PROGRAM Log_Diverts_P2150
VAR
	r_DivertExtend			: ARRAY [1..16] OF R_TRIG;
	f_DivertExtend			: ARRAY [1..16] OF F_TRIG;
	r_ConfirmPE				: ARRAY [1..16] OF R_TRIG;
	f_ConfirmPE				: ARRAY [1..16] OF F_TRIG;
	sMessage				: STRING;
END_VAR

// Divert 1
r_DivertExtend[1](CLK := Sorter.aSorterDiverts_P2150[1].Output1);
f_DivertExtend[1](CLK := Sorter.aSorterDiverts_P2150[1].Output1);

IF r_DivertExtend[1].Q THEN
	IF .nDivertLogEnable.DIVERT1 THEN
		ADSLOGSTR( msgCtrlMask := ADSLOG_MSGTYPE_HINT OR ADSLOG_MSGTYPE_LOG
			, msgFmtStr := 'Extend Divert 1 : %s'
			, strArg := UDINT_TO_STRING(Sorter.st_SorterEncoder_P2150.CurrentCount)); 
	END_IF;
END_IF
IF f_DivertExtend[1].Q THEN
	IF .nDivertLogEnable.DIVERT1 THEN
		ADSLOGSTR( msgCtrlMask := ADSLOG_MSGTYPE_HINT OR ADSLOG_MSGTYPE_LOG
			, msgFmtStr := 'Retract Divert 1 : %s'
			, strArg := UDINT_TO_STRING(Sorter.st_SorterEncoder_P2150.CurrentCount)); 
	END_IF;
END_IF

// Confirm 1
r_ConfirmPE[1](CLK := Sorter.aSorterDiverts_P2150[1].ConfirmPE);
f_ConfirmPE[1](CLK := Sorter.aSorterDiverts_P2150[1].ConfirmPE);

IF r_ConfirmPE[1].Q THEN
	IF .nDivertLogEnable.CONFIRM1 THEN
		ADSLOGSTR( msgCtrlMask := ADSLOG_MSGTYPE_HINT OR ADSLOG_MSGTYPE_LOG
			, msgFmtStr := 'Confirm PE 1 Blocked: %s'
			, strArg := UDINT_TO_STRING(Sorter.st_SorterEncoder_P2150.CurrentCount)); 
	END_IF;
END_IF
IF f_ConfirmPE[1].Q THEN
	IF .nDivertLogEnable.CONFIRM1 THEN
		ADSLOGSTR( msgCtrlMask := ADSLOG_MSGTYPE_HINT OR ADSLOG_MSGTYPE_LOG
			, msgFmtStr := 'Confirm PE 1 Clear: %s'
			, strArg := UDINT_TO_STRING(Sorter.st_SorterEncoder_P2150.CurrentCount)); 
	END_IF;
END_IF

// Divert 2
r_DivertExtend[2](CLK := Sorter.aSorterDiverts_P2150[2].Output1);
f_DivertExtend[2](CLK := Sorter.aSorterDiverts_P2150[2].Output1);

IF r_DivertExtend[2].Q THEN
	IF .nDivertLogEnable.DIVERT2 THEN
		ADSLOGSTR( msgCtrlMask := ADSLOG_MSGTYPE_HINT OR ADSLOG_MSGTYPE_LOG
			, msgFmtStr := 'Extend Divert 2: %s'
			, strArg := UDINT_TO_STRING(Sorter.st_SorterEncoder_P2150.CurrentCount)); 
	END_IF;
END_IF
IF f_DivertExtend[2].Q THEN
	IF .nDivertLogEnable.DIVERT2 THEN
		ADSLOGSTR( msgCtrlMask := ADSLOG_MSGTYPE_HINT OR ADSLOG_MSGTYPE_LOG
			, msgFmtStr := 'Retract Divert 2: %s'
			, strArg := UDINT_TO_STRING(Sorter.st_SorterEncoder_P2150.CurrentCount)); 
	END_IF;
END_IF

// Confirm 2
r_ConfirmPE[2](CLK := Sorter.aSorterDiverts_P2150[2].ConfirmPE);
f_ConfirmPE[2](CLK := Sorter.aSorterDiverts_P2150[2].ConfirmPE);

IF r_ConfirmPE[2].Q THEN
	IF .nDivertLogEnable.CONFIRM2 THEN
		ADSLOGSTR( msgCtrlMask := ADSLOG_MSGTYPE_HINT OR ADSLOG_MSGTYPE_LOG
			, msgFmtStr := 'Confirm PE 2 Blocked: %s'
			, strArg := UDINT_TO_STRING(Sorter.st_SorterEncoder_P2150.CurrentCount)); 
	END_IF;
END_IF
IF f_ConfirmPE[2].Q THEN
	IF .nDivertLogEnable.CONFIRM2 THEN
		ADSLOGSTR( msgCtrlMask := ADSLOG_MSGTYPE_HINT OR ADSLOG_MSGTYPE_LOG
			, msgFmtStr := 'Confirm PE 2 Clear: %s'
			, strArg := UDINT_TO_STRING(Sorter.st_SorterEncoder_P2150.CurrentCount)); 
	END_IF
END_IF

// Sorter Discharge "Divert"
// Divert 3
r_DivertExtend[3](CLK := Sorter.aSorterDiverts_P2150[3].Output1);
f_DivertExtend[3](CLK := Sorter.aSorterDiverts_P2150[3].Output1);

IF r_DivertExtend[3].Q THEN
	IF .nDivertLogEnable.DIVERT3 THEN
		ADSLOGSTR( msgCtrlMask := ADSLOG_MSGTYPE_HINT OR ADSLOG_MSGTYPE_LOG
			, msgFmtStr := 'Extend Divert 3: %s'
			, strArg := UDINT_TO_STRING(Sorter.st_SorterEncoder_P2150.CurrentCount)); 
	END_IF;
END_IF
IF f_DivertExtend[3].Q THEN
	IF .nDivertLogEnable.DIVERT3 THEN
		ADSLOGSTR( msgCtrlMask := ADSLOG_MSGTYPE_HINT OR ADSLOG_MSGTYPE_LOG
			, msgFmtStr := 'Retract Divert 3: %s'
			, strArg := UDINT_TO_STRING(Sorter.st_SorterEncoder_P2150.CurrentCount)); 
	END_IF;
END_IF

// Confirm 3
r_ConfirmPE[3](CLK := Sorter.aSorterDiverts_P2150[3].ConfirmPE);
f_ConfirmPE[3](CLK := Sorter.aSorterDiverts_P2150[3].ConfirmPE);

IF r_ConfirmPE[3].Q THEN
	IF .nDivertLogEnable.CONFIRM3 THEN
		ADSLOGSTR( msgCtrlMask := ADSLOG_MSGTYPE_HINT OR ADSLOG_MSGTYPE_LOG
			, msgFmtStr := 'Confirm PE 3 Blocked: %s'
			, strArg := UDINT_TO_STRING(Sorter.st_SorterEncoder_P2150.CurrentCount)); 
	END_IF;
END_IF
IF f_ConfirmPE[3].Q THEN
	IF .nDivertLogEnable.CONFIRM3 THEN
		ADSLOGSTR( msgCtrlMask := ADSLOG_MSGTYPE_HINT OR ADSLOG_MSGTYPE_LOG
			, msgFmtStr := 'Confirm PE 3 Clear: %s'
			, strArg := UDINT_TO_STRING(Sorter.st_SorterEncoder_P2150.CurrentCount)); 
	END_IF
END_IF

// Sorter Discharge "Divert"
// Divert 4
r_DivertExtend[4](CLK := Sorter.aSorterDiverts_P2150[4].Output1);
f_DivertExtend[4](CLK := Sorter.aSorterDiverts_P2150[4].Output1);

IF r_DivertExtend[4].Q THEN
	IF .nDivertLogEnable.DIVERT4 THEN
		ADSLOGSTR( msgCtrlMask := ADSLOG_MSGTYPE_HINT OR ADSLOG_MSGTYPE_LOG
			, msgFmtStr := 'Extend Divert 4: %s'
			, strArg := UDINT_TO_STRING(Sorter.st_SorterEncoder_P2150.CurrentCount)); 
	END_IF;
END_IF
IF f_DivertExtend[4].Q THEN
	IF .nDivertLogEnable.DIVERT4 THEN
		ADSLOGSTR( msgCtrlMask := ADSLOG_MSGTYPE_HINT OR ADSLOG_MSGTYPE_LOG
			, msgFmtStr := 'Retract Divert 4: %s'
			, strArg := UDINT_TO_STRING(Sorter.st_SorterEncoder_P2150.CurrentCount)); 
	END_IF;
END_IF

// Confirm 4
r_ConfirmPE[4](CLK := Sorter.aSorterDiverts_P2150[4].ConfirmPE);
f_ConfirmPE[4](CLK := Sorter.aSorterDiverts_P2150[4].ConfirmPE);

IF r_ConfirmPE[4].Q THEN
	IF .nDivertLogEnable.CONFIRM4 THEN
		ADSLOGSTR( msgCtrlMask := ADSLOG_MSGTYPE_HINT OR ADSLOG_MSGTYPE_LOG
			, msgFmtStr := 'Confirm PE 4 Blocked: %s'
			, strArg := UDINT_TO_STRING(Sorter.st_SorterEncoder_P2150.CurrentCount)); 
	END_IF;
END_IF
IF f_ConfirmPE[4].Q THEN
	IF .nDivertLogEnable.CONFIRM4 THEN
		ADSLOGSTR( msgCtrlMask := ADSLOG_MSGTYPE_HINT OR ADSLOG_MSGTYPE_LOG
			, msgFmtStr := 'Confirm PE 4 Clear: %s'
			, strArg := UDINT_TO_STRING(Sorter.st_SorterEncoder_P2150.CurrentCount)); 
	END_IF
END_IF	

// Sorter Discharge "Divert"
// Divert 5
r_DivertExtend[5](CLK := Sorter.aSorterDiverts_P2150[5].Output1);
f_DivertExtend[5](CLK := Sorter.aSorterDiverts_P2150[5].Output1);

IF r_DivertExtend[5].Q THEN
	IF .nDivertLogEnable.DIVERT5 THEN
		ADSLOGSTR( msgCtrlMask := ADSLOG_MSGTYPE_HINT OR ADSLOG_MSGTYPE_LOG
			, msgFmtStr := 'Extend Divert 5: %s'
			, strArg := UDINT_TO_STRING(Sorter.st_SorterEncoder_P2150.CurrentCount)); 
	END_IF;
END_IF
IF f_DivertExtend[5].Q THEN
	IF .nDivertLogEnable.DIVERT5 THEN
		ADSLOGSTR( msgCtrlMask := ADSLOG_MSGTYPE_HINT OR ADSLOG_MSGTYPE_LOG
			, msgFmtStr := 'Retract Divert 5: %s'
			, strArg := UDINT_TO_STRING(Sorter.st_SorterEncoder_P2150.CurrentCount)); 
	END_IF;
END_IF

// Confirm 5
r_ConfirmPE[5](CLK := Sorter.aSorterDiverts_P2150[5].ConfirmPE);
f_ConfirmPE[5](CLK := Sorter.aSorterDiverts_P2150[5].ConfirmPE);

IF r_ConfirmPE[5].Q THEN
	IF .nDivertLogEnable.CONFIRM5 THEN
		ADSLOGSTR( msgCtrlMask := ADSLOG_MSGTYPE_HINT OR ADSLOG_MSGTYPE_LOG
			, msgFmtStr := 'Confirm PE 5 Blocked: %s'
			, strArg := UDINT_TO_STRING(Sorter.st_SorterEncoder_P2150.CurrentCount)); 
	END_IF;
END_IF
IF f_ConfirmPE[5].Q THEN
	IF .nDivertLogEnable.CONFIRM5 THEN
		ADSLOGSTR( msgCtrlMask := ADSLOG_MSGTYPE_HINT OR ADSLOG_MSGTYPE_LOG
			, msgFmtStr := 'Confirm PE 5 Clear: %s'
			, strArg := UDINT_TO_STRING(Sorter.st_SorterEncoder_P2150.CurrentCount)); 
	END_IF
END_IF

END_PROGRAM

(* stored: Version 1.1.0.1, ProductVersion 3.1.4024.4
   POU Log_Diverts_P2150: Id {96d68961-3ed5-4ea2-ae0e-09cce6fa5594}, SpecialFunc None *)
